// TwinCAT 3 PLC project PLC1
// ProgramVersion: 3.1.4024.12
// libraries:
//   Tc2_Standard, * (Beckhoff Automation GmbH)
//   Tc2_System, * (Beckhoff Automation GmbH)
//   Tc3_Module, * (Beckhoff Automation GmbH)
// project tree:
//   Diagrams/ Class Diagram.TcCD (not stored)
//   FBs/ FB_Generator.TcPOU (not stored), FB_GeneratorEX.TcPOU (not stored)
//   / PlcTask.TcTTO
//   POUs/ MAIN.TcPOU
// real-time tasks:
//   TASK PlcTask: cycle T#10ms, priority 20, ADS port 350

CONFIGURATION PLC1
    RESOURCE PLC ON TwinCAT3
        TASK PlcTask(INTERVAL := T#10ms, PRIORITY := 20);
        PROGRAM MAIN WITH PlcTask : MAIN;
    END_RESOURCE
END_CONFIGURATION

// ---- POUs/MAIN.TcPOU
PROGRAM MAIN
VAR
	// Instance of Generator 1
	fbGenerator1 :FB_Generator;	
	// Instance of Generator 2
	fbGenerator2 :FB_GeneratorEX;	
	
	// Status of flasher 1
	Flasher1: BOOL;
	// Status of flasher 2
	Flasher2: BOOL;
END_VAR

// Set the cycletime property for the class
fbGenerator1.Cycletime := T#2S;
fbGenerator2.Cycletime := T#2S;

// Call the flasher method
Flasher1 := fbGenerator1.Flash();
Flasher2 := fbGenerator2.Flash();

END_PROGRAM
